FUNCTION_BLOCK tool_changeover
VAR_INPUT 
	// LREAL
	actual_pos                 : LREAL;
	actual_vel                 : LREAL;
	target_work_pos            : LREAL;
	target_home_pos            : LREAL;
	target_vel_from_hmi        : LREAL;
	SERVO_TOL_CHECK_OFFSET_POS : LREAL;	
	//INT
	station_number             : INT;
	mover_number               : INT;
	no_of_mover_present        : INT;
	model_selected             : INT;
	
	//BOOL
	tool_unloading_start       : BOOL;
	tool_loading_start         : BOOL;
	error_active               : BOOL;
	station_in_auto            : BOOL;
	station_in_home            : BOOL;
	absoulte_move_done         : BOOL;
	tool_6_3_present           : BOOL;
	tool_7_89_present          : BOOL;
	fb_reset                   : BOOL;
    operator_ack               : BOOL;
	
END_VAR                        

VAR_OUTPUT PERSISTENT
	tool_changer_over_complete : BOOL;
	tool_disengage             : BOOL;
	tool_engagae               : BOOL;
	tool_loading_complete		: BOOL;
	tool_unloading_complete    : BOOL;
	servo_move_abs             : BOOL;
	tool_loading_failed        : BOOL;
	unloading_status           : STRING;
	loading_status             : STRING;
	
	target_pos_to_servo        : LREAL;
	target_vel_to_servo        : LREAL;
	
END_VAR

VAR PERSISTENT
	//INT
	Unloading_Sequence         : INT;
	Loading_Sequence           : INT;
	model_present              : INT;
	
	// BOOL
	target_pos_reached		   : BOOL;
	engaged_check              : BOOL;
	unloading_started          : BOOL; 
	loading_started            : BOOL;
	disengage_check            : BOOL;
	//TIMER
	disengage_timer            :ton;
	engage_timer               :ton;
	disengae_timer             :TON;
	
	
END_VAR

VAR
	SERVO_WRK_POS				: BOOL;
	SERVO_HME_POS				: BOOL;
	SERVO_TOL_CHCK_POS          : BOOL;
	dis: BOOL;
END_VAR
VAR_IN_OUT
	
END_VAR

                                    ////////////////////////////////////// GENERAL SEQUENCE //////////////////////////////////////

IF (error_active AND station_in_auto) THEN
	tool_disengage             := FALSE;
	tool_engagae               := FALSE;
	servo_move_abs             := FALSE;
	unloading_status           := 'error active clear error';
	
ELSIF  NOT error_active AND NOT station_in_auto THEN
		unloading_status       := 'station is not in auto';
		
ELSIF NOT error_active AND station_in_auto AND station_in_home AND NOT unloading_started AND NOT loading_started THEN
	  Unloading_Sequence        := 0;
	  loading_Sequence          := 0;
	  
	  IF tool_changer_over_complete THEN
	  tool_changer_over_complete := FALSE;
	  END_IF
END_IF

                         ////////////////////////////////////////// block complete reset //////////////////////////////////////////
						 
IF fb_reset THEN
	tool_changer_over_complete := FALSE;
	tool_disengage             := false;
	tool_engagae               := false;
	tool_loading_complete      := false;
	tool_unloading_complete    := false;
	servo_move_abs             := FALSE;
	SERVO_WRK_POS			   := FALSE;
	SERVO_HME_POS			   := FALSE;
	SERVO_TOL_CHCK_POS         := FALSE;
	engaged_check              := FALSE;
	unloading_started          := FALSE;	
	unloading_status           := 'block reseted';
	loading_status             := 'block reseted';
	target_pos_to_servo        := 0.0;
	target_vel_to_servo		   := 0.0;
    Unloading_Sequence         := 0;
    loading_Sequence           := 0;	
END_IF 

               ////////////////////////////////////////////////////// model selected ///////////////////////////////////////////////////////////
			   
// model number = 1 then tool for 6.3 present
// model number = 2 then tool for 7.89 present	
	   
IF tool_6_3_present AND NOT tool_7_89_present THEN
	  model_present :=1;
ELSIF tool_7_89_present AND NOT tool_6_3_present THEN
	  model_present :=2;
END_IF


                            ////////////////////////////////////// UNLOADING SEQUENCE //////////////////////////////////////////
							
CASE Unloading_Sequence OF
	
     0: IF NOT tool_loading_complete  AND NOT tool_unloading_complete  AND	tool_unloading_start THEN          // check tool change over start command
		       unloading_started := TRUE;
               Unloading_Sequence := 10;
	    ELSIF NOT tool_unloading_start THEN
	          unloading_status := 'waiting for tool unloading start command';
		ELSIF NOT tool_unloading_complete THEN
			 unloading_status := 'previous unloading complete bit is not reseted';
		ELSIF NOT tool_loading_complete THEN
			 unloading_status := 'previous loading complete bit is not reseted';	 
	 END_IF
	 
	 
	 10: IF model_selected = model_present THEN
		   Unloading_Sequence  :=  60;
		ELSIF model_selected <> model_present THEN
			Unloading_Sequence  :=  20;
	    END_IF
	 
     20: target_pos_to_servo := target_work_pos ;                                                              // moving target position and velocity to servo 
         target_vel_to_servo := target_vel_from_hmi ;
		 
		 IF target_pos_to_servo = target_work_pos AND target_vel_to_servo = target_vel_from_hmi THEN
			 servo_move_abs      := TRUE;
			 unloading_status    := ' target position and velocity to servo moved ';
			 Unloading_Sequence  :=  30;
	     ELSIF target_pos_to_servo <> target_work_pos OR target_vel_to_servo <> target_vel_from_hmi THEN	
		      unloading_status   := ' target position or velocity to servo not moved ';
		 END_IF
		 
	 30: IF  absoulte_move_done AND SERVO_WRK_POS  THEN
		 
		     servo_move_abs := FALSE;
             tool_disengage := TRUE;
			 Unloading_Sequence  := 40;
			 
		 ELSIF NOT absoulte_move_done AND SERVO_WRK_POS THEN 
			   unloading_status   := ' waiting for absolute done ';
	     ELSIF 	absoulte_move_done AND NOT SERVO_WRK_POS THEN 
			 unloading_status   := ' waiting target pos reached fb ';		 
		 END_IF 	 
		
	 40: IF disengage_timer.Q THEN
		    target_pos_to_servo := target_work_pos - SERVO_TOL_CHECK_OFFSET_POS;                                                              
            target_vel_to_servo := target_vel_from_hmi ;
			
             IF target_pos_to_servo = target_work_pos- SERVO_TOL_CHECK_OFFSET_POS AND target_vel_to_servo = target_vel_from_hmi THEN
			  servo_move_abs      := TRUE;
			  Unloading_Sequence  := 50;
			  unloading_status    := ' target position and velocity to servo moved ';
			  
			  ELSIF target_pos_to_servo <> target_work_pos- SERVO_TOL_CHECK_OFFSET_POS OR target_vel_to_servo <> target_vel_from_hmi THEN
				     unloading_status   := ' target position or velocity to servo not moved ';
		     END_IF
			
		ELSIF NOT disengage_timer.Q THEN
			  unloading_status   := ' waiting for 5s  ';
	    END_IF
		
		
     50: IF absoulte_move_done  AND SERVO_TOL_CHCK_POS THEN
		    servo_move_abs := FALSE;
		    Unloading_Sequence  := 60;
			
		ELSIF NOT absoulte_move_done AND SERVO_TOL_CHCK_POS THEN 
			   unloading_status   := ' waiting for absolute done ';
			   
	     ELSIF 	absoulte_move_done AND NOT SERVO_TOL_CHCK_POS THEN 
			 unloading_status   := ' waiting target pos reached fb ';	
	 END_IF

  
	 60: IF  model_present = 1  THEN
		     IF NOT tool_6_3_present THEN
                    tool_disengage := FALSE;
			        target_pos_to_servo := target_home_pos;                                                              
                    target_vel_to_servo := target_vel_from_hmi;
			        unloading_status   := ' tool disengaged ';	
			     IF target_pos_to_servo = target_home_pos AND target_vel_to_servo = target_vel_from_hmi THEN
			      servo_move_abs      := TRUE;
			      Unloading_Sequence  := 70;  
			     ELSIF target_pos_to_servo <> target_home_pos OR target_vel_to_servo <> target_vel_from_hmi THEN
	                 unloading_status   := ' target position or velocity to servo not moved ';
		         END_IF	  
 
			 ELSIF  tool_6_3_present THEN
				    unloading_status   := ' tool not disengaged ';
			 END_IF 
			 
		 ELSIF  model_present = 2 THEN
			   IF NOT  tool_7_89_present THEN
				       tool_disengage := FALSE;
			           target_pos_to_servo := target_home_pos;                                                              
                       target_vel_to_servo := target_vel_from_hmi;
			           unloading_status   := ' tool disengaged ';  
			       IF target_pos_to_servo = target_home_pos AND target_vel_to_servo = target_vel_from_hmi THEN
			          servo_move_abs      := TRUE;
			          Unloading_Sequence  := 70;
			        ELSIF target_pos_to_servo <> target_home_pos OR target_vel_to_servo <> target_vel_from_hmi THEN
	                  unloading_status   := ' target position or velocity to servo not moved ';
		           END_IF
			   
			   ELSIF  tool_7_89_present THEN
				       unloading_status   := ' tool not disengaged ';
			   
			   END_IF
	 
		 END_IF

		
     70: IF  absoulte_move_done AND SERVO_HME_POS  THEN
     		 
     		     servo_move_abs         := FALSE;
     	         Unloading_Sequence     := 80;
				 
         ELSIF NOT absoulte_move_done AND SERVO_HME_POS THEN 
     			   unloading_status   := ' waiting for absolute done ';
     			   
     	 ELSIF 	absoulte_move_done AND NOT SERVO_HME_POS THEN 
     			 unloading_status   := ' waiting target pos reached fb ';
     		 
     	 END_IF

     80: IF  NOT tool_7_89_present AND NOT tool_6_3_present THEN
             tool_unloading_complete:= TRUE;
             model_present :=0;
		 END_IF
		 
END_CASE


                               ////////////////////////////////////// LOADING SEQUENCE /////////////////////////////////////////////
							   
CASE loading_sequence OF
	
	0: IF 	tool_loading_start AND tool_unloading_complete AND model_present = 0 AND Unloading_Sequence = 80 THEN
		    loading_Sequence := 10;
	    ELSIF NOT 	tool_loading_start AND tool_unloading_complete AND model_present = 0 THEN
	          loading_status := 'waiting for tool chageover start command';
	    ELSIF tool_loading_start AND NOT tool_unloading_complete AND model_present = 0 THEN
		       loading_status := 'waiting for tool unloding complete feedback';
		ELSIF tool_loading_start AND  tool_unloading_complete AND  model_present <> 0	THEN
              loading_status := 'model present is not equal to 0 ';
	 END_IF
	 
     10: target_pos_to_servo := target_work_pos ;                                                              // moving work position and velocity to servo 
         target_vel_to_servo := target_vel_from_hmi ;
		 tool_disengage      := TRUE ;
		 
		 IF target_pos_to_servo = target_work_pos AND target_vel_to_servo = target_vel_from_hmi THEN
			 servo_move_abs      := TRUE;
			 loading_status    := ' target position and velocity to servo moved ';
			 loading_Sequence  :=  20;
	     ELSIF target_pos_to_servo <> target_work_pos OR target_vel_to_servo <> target_vel_from_hmi THEN	
		      loading_status   := ' target position or velocity to servo not moved ';
		 END_IF
		 
	 20: IF  absoulte_move_done AND SERVO_WRK_POS  THEN
		 
		     servo_move_abs := FALSE;
			 engaged_check  := TRUE ;
			 tool_disengage := FALSE ;
			 tool_engagae   := TRUE;
			 loading_Sequence  := 30;
			 
		 ELSIF NOT absoulte_move_done AND SERVO_WRK_POS THEN 
			   loading_status   := ' waiting for absolute done ';
	     ELSIF 	absoulte_move_done AND NOT SERVO_WRK_POS THEN 
			 loading_status   := ' waiting target pos reached fb ';		 
		 END_IF 	 
		
	 30: IF engage_timer.q THEN
		    target_pos_to_servo := target_work_pos - SERVO_TOL_CHECK_OFFSET_POS;          // moving enage position and velocity to servo                                                     
            target_vel_to_servo := target_vel_from_hmi ;
			engaged_check       := FALSE;
             IF target_pos_to_servo = target_work_pos- SERVO_TOL_CHECK_OFFSET_POS AND target_vel_to_servo = target_vel_from_hmi THEN
			  servo_move_abs      := TRUE;
			  loading_Sequence  := 40;
			 ELSIF target_pos_to_servo <> target_work_pos- SERVO_TOL_CHECK_OFFSET_POS OR target_vel_to_servo <> target_vel_from_hmi THEN 
				   loading_status   := ' target position or velocity to servo not moved ';
		     END_IF
			
	    END_IF
		
		
	 
	 40: IF  absoulte_move_done AND SERVO_TOL_CHCK_POS  THEN
		     servo_move_abs := FALSE;
			 loading_Sequence  := 50;
		 ELSIF NOT absoulte_move_done AND SERVO_TOL_CHCK_POS THEN 
			   loading_status   := ' waiting for absolute done ';   
	     ELSIF 	absoulte_move_done AND NOT SERVO_TOL_CHCK_POS THEN 
			 loading_status   := ' waiting target pos reached fb ';	
		 END_IF

	         
	 
		 50: IF model_selected=1 THEN                       // moving home position and velocity to servo  
                   IF tool_6_3_present AND  model_present = 1 THEN
				   target_pos_to_servo := target_home_pos;                                                              
                   target_vel_to_servo := target_vel_from_hmi;
			 
			        IF target_pos_to_servo = target_home_pos AND target_vel_to_servo = target_vel_from_hmi THEN
			           servo_move_abs      := TRUE;
			           loading_Sequence  := 60;
					   
					ELSIF target_pos_to_servo <>  target_home_pos AND target_vel_to_servo <> target_vel_from_hmi THEN  
                            loading_status   := ' target position or velocity to servo not moved '; 
		             END_IF
				   ELSIF NOT (tool_6_3_present AND tool_7_89_present) OR  model_present <> 1 THEN
	                     loading_status   :='tool not engaged';
					ELSIF (NOT tool_6_3_present AND tool_7_89_present) AND  model_present <> 1 THEN
						   loading_Sequence  := 101;
				END_IF
				
             ELSIF model_selected=2 THEN
				   IF tool_7_89_present AND  model_present = 2 THEN
					  target_pos_to_servo := target_home_pos;                                                              
                      target_vel_to_servo := target_vel_from_hmi;
			 
			          IF target_pos_to_servo = target_home_pos AND target_vel_to_servo = target_vel_from_hmi THEN
			           servo_move_abs      := TRUE;
			           loading_Sequence  := 60;
					  ELSIF target_pos_to_servo <>  target_home_pos AND target_vel_to_servo <> target_vel_from_hmi THEN  
                            loading_status   := ' target position or velocity to servo not moved '; 
		             END_IF
					 
					 ELSIF (  tool_7_89_present AND tool_6_3_present ) OR  model_present <> 2 THEN
						   loading_status   :='tool not engaged';
						   
					 ELSIF ( tool_6_3_present AND NOT tool_7_89_present) AND  model_present <> 2 THEN
						   loading_Sequence  := 101;
	   
                   END_IF
		    END_IF 
		
		
     60: IF  absoulte_move_done AND SERVO_HME_POS  THEN
     		     servo_move_abs         := FALSE;
     	         loading_Sequence       := 70;
				 
         ELSIF NOT absoulte_move_done AND SERVO_HME_POS THEN 
     			   loading_status   := ' waiting for absolute done ';
     			   
     	 ELSIF 	absoulte_move_done AND NOT SERVO_HME_POS THEN 
     			 loading_status   := ' waiting target pos reached fb ';
     		 
     	 END_IF

     70:  tool_loading_complete:= TRUE;
	      loading_Sequence     := 80;
	 
     80: IF  tool_loading_complete AND tool_unloading_complete THEN
		 unloading_started := FALSE;
		 loading_started   := FALSE;
		 tool_changer_over_complete := TRUE;
		 tool_engagae   := FALSE;
	     END_IF
	  
	  101: IF  operator_ack THEN
		       target_pos_to_servo := target_work_pos ;                                                               
               target_vel_to_servo := target_vel_from_hmi ;
			  IF target_pos_to_servo = target_work_pos AND target_vel_to_servo = target_vel_from_hmi THEN
			     servo_move_abs      := TRUE;
			     loading_status    := ' target position and velocity to servo moved ';
			     loading_Sequence  :=  110;
	         ELSIF target_pos_to_servo <> target_work_pos OR target_vel_to_servo <> target_vel_from_hmi THEN	
		      loading_status   := ' target position or velocity to servo not moved ';
		     END_IF
	     END_IF
	  
	  110: IF absoulte_move_done AND SERVO_WRK_POS  THEN
		     servo_move_abs := FALSE;
			 tool_disengage := TRUE ;
			 disengage_check  := TRUE ;
			 tool_engagae   := FALSE;
			 loading_Sequence  := 120;
			 
		 ELSIF NOT absoulte_move_done AND SERVO_WRK_POS THEN 
			   loading_status   := ' waiting for absolute done ';
	     ELSIF 	absoulte_move_done AND NOT SERVO_WRK_POS THEN 
			 loading_status   := ' waiting target pos reached fb ';		 
		 END_IF 	 
	  
	  120:  IF engage_timer.q THEN
		       target_pos_to_servo := target_work_pos - SERVO_TOL_CHECK_OFFSET_POS;          // moving enage position and velocity to servo                                                     
               target_vel_to_servo := target_vel_from_hmi ;
			   disengage_check       := FALSE;
               IF target_pos_to_servo = target_work_pos- SERVO_TOL_CHECK_OFFSET_POS AND target_vel_to_servo = target_vel_from_hmi THEN
			      servo_move_abs      := TRUE;
			      loading_Sequence  := 130;
			   ELSIF target_pos_to_servo <> target_work_pos- SERVO_TOL_CHECK_OFFSET_POS OR target_vel_to_servo <> target_vel_from_hmi THEN 
				   loading_status   := ' target position or velocity to servo not moved ';
		       END_IF
	        END_IF
			
	  130:  IF NOT (tool_6_3_present AND tool_7_89_present) THEN
		         target_pos_to_servo := target_home_pos;                                                              
                 target_vel_to_servo := target_vel_from_hmi;
			     IF target_pos_to_servo = target_home_pos AND target_vel_to_servo = target_vel_from_hmi THEN
			        servo_move_abs      := TRUE;
			        loading_Sequence  := 140;
				 ELSIF target_pos_to_servo <>  target_home_pos AND target_vel_to_servo <> target_vel_from_hmi THEN  
                       loading_status   := ' target position or velocity to servo not moved '; 
		         END_IF
	        END_IF
			
	 140: 	 IF  absoulte_move_done AND SERVO_HME_POS  THEN
            	     servo_move_abs         := FALSE;
                     loading_Sequence       := 150;
            		 
             ELSIF NOT absoulte_move_done AND SERVO_HME_POS THEN 
            		   loading_status   := ' waiting for absolute done ';
            		   
             ELSIF 	absoulte_move_done AND NOT SERVO_HME_POS THEN 
            		 loading_status   := ' waiting target pos reached fb ';
            	 
             END_IF
			 
      150:   tool_loading_failed := TRUE;
	          
END_CASE


                                                           //////////////////  timer for logic //////////////////////////////// j
														   
disengage_timer(IN:= tool_disengage , PT:= T#5S, Q=> , ET=> );
engage_timer(IN:= engaged_check , PT:= T#5S, Q=> , ET=> );
disengae_timer(IN:= disengage_check , PT:= , Q=> , ET=> );


// #################################	IN RANGE 		##############################


SERVO_WRK_POS		:=In_Range(value:=actual_pos, setvalue:=target_work_pos, tolerance:=0.2 );
SERVO_HME_POS		:=In_Range(value:=actual_pos, setvalue:=target_home_pos, tolerance:=0.2 );
SERVO_TOL_CHCK_POS	:=In_Range(value:=actual_pos, setvalue:=target_work_pos-SERVO_TOL_CHECK_OFFSET_POS, tolerance:=0.2 );

END_FUNCTION_BLOCK

(* stored: Version 1.1.0.1, ProductVersion 3.1.4024.11
   POU tool_changeover: Id {b828edc9-90a1-4354-aeee-747e8c699690}, SpecialFunc None *)
